PROGRAM MAIN
VAR
END_VAR

prg_PotentioMeter();
prg_DynamischVerschalen();

END_PROGRAM

(* stored: Version 1.1.0.1, ProductVersion 3.1.4024.15
   POU MAIN: Id {34531326-9eb4-4723-9f4e-42b2ad864a36}, SpecialFunc None *)
